// SIMATIC S7-200 SMART project (STEP 7-Micro/WIN SMART), CPU SR20

SYMBOL_TABLE System Symbols
Always_On        SM0.0    // Always ON
END_SYMBOL_TABLE

ORGANIZATION_BLOCK MAIN:OB1
TITLE=Program Comments
BEGIN
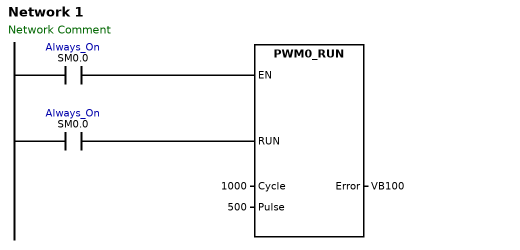
Network 1
// Network Comment
LD     Always_On:SM0.0
=      L60.0
LD     Always_On:SM0.0
=      L63.7
LD     L60.0
CALL   PWM0_RUN:SBR1, L63.7, 1000, 500, VB100
END_ORGANIZATION_BLOCK

SUBROUTINE_BLOCK SBR_0:SBR0
TITLE=Subroutine Comments
BEGIN
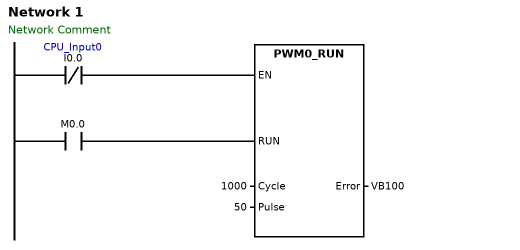
Network 1
// Network Comment
LDN    CPU_Input0:I0.0
=      L60.0
LD     M0.0
=      L63.7
LD     L60.0
CALL   PWM0_RUN:SBR1, L63.7, 1000, 50, VB100
END_SUBROUTINE_BLOCK

// SBR1: protected block, not included

DATA_BLOCK_TAB Page_1
BEGIN
V100     123
END_DATA_BLOCK_TAB
